// TIA Portal project "llenado Automatico" (V18)
// Sistema de llenado automatico de cajas

(* hardware
DEVICE "S7-1200 station_1"  S7-1200 Station
   slot 0: "Rack_0"  S7-1200 Rack  Rack  V1.0
   slot 1: "PLC_1"  CPU 1212C AC/DC/Rly  6ES7 212-1BE40-0XB0  V4.6
*)

// ===== PLC "PLC_1"  CPU 1212C AC/DC/Rly =====

VAR_GLOBAL   // PLC tag table "OUTPUTS"
   "CONVEYOR" AT %Q0.0 : Bool;
   "SOLENOID" AT %Q0.1 : Bool;
   "RUN_INDICATOR" AT %Q0.2 : Bool;
   "STANDBY_INDICATOR" AT %Q0.3 : Bool;
   "FULLBOX_INDICATOR" AT %Q0.4 : Bool;
END_VAR

VAR_GLOBAL   // PLC tag table "INPUTS"
   "START_PROCESS" AT %I0.0 : Bool;
   "STOP_PROCESS" AT %I0.1 : Bool;
   "LEVEL_BOX_SENSOR" AT %I0.3 : Bool;
   "BOX_POSITION_SENSOR" AT %I0.4 : Bool;
   "EMERGENCY_STOP" AT %I0.2 : Bool;
END_VAR

// folder: GLOBAL VARIABLES

DATA_BLOCK "GLOBAL_VARIABLES"   // DB1
TITLE = Global Variables
{ S7_Optimized_Access := 'TRUE' }
AUTHOR : Stiven Perez Mora
VERSION : 0.1
   VAR
      SET_RESET_PROCESS : Bool;
   END_VAR
BEGIN
END_DATA_BLOCK

// folder: (top level)

FUNCTION "START_STOP_PROCESS" : Void   // FC1, LAD
TITLE = Start - Stop process
{ S7_Optimized_Access := 'TRUE' }
AUTHOR : Stiven Perez Mora
VERSION : 0.1
BEGIN

REGION Network 1: START - STOP ALL THE PROCESS
   // CONDITIONS TO START STOP ALL THE PROCESS
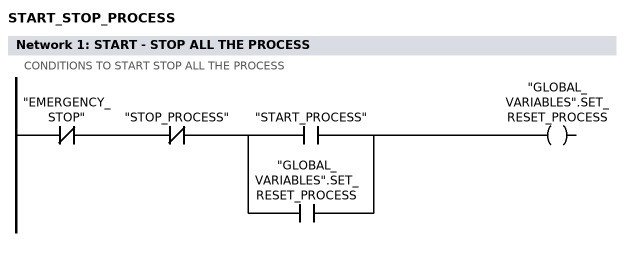
   RUNG wire#powerrail
      I_Contact( "EMERGENCY_STOP" )
      I_Contact( "STOP_PROCESS" )
      wire#w1
      Contact( "START_PROCESS" )
      wire#w2
      Coil( "GLOBAL_VARIABLES".SET_RESET_PROCESS )
   END_RUNG
   RUNG wire#w1
      Contact( "GLOBAL_VARIABLES".SET_RESET_PROCESS )
   END_RUNG wire#w2
   // the same network as SCL:
   "GLOBAL_VARIABLES".SET_RESET_PROCESS := NOT "EMERGENCY_STOP" AND NOT "STOP_PROCESS" AND ("START_PROCESS" OR "GLOBAL_VARIABLES".SET_RESET_PROCESS);
END_REGION
END_FUNCTION

ORGANIZATION_BLOCK "Main"   // OB1, LAD, ProgramCycle
TITLE = "Main Program Sweep (Cycle)"
{ S7_Optimized_Access := 'TRUE' }
VERSION : 0.1
   VAR_INPUT
      Initial_Call : Bool;   // Initial call of this OB
      Remanence : Bool;   // =True, if remanent data are available
   END_VAR
BEGIN
END_ORGANIZATION_BLOCK